// TwinCAT 3 PLC project PLC
// ProgramVersion: 3.1.4023.0
// libraries:
//   Tc2_Standard, * (Beckhoff Automation GmbH)
//   Tc2_System, * (Beckhoff Automation GmbH)
//   Tc3_Module, * (Beckhoff Automation GmbH)
// project tree:
//   DUTs/ ST_ControlBits.TcDUT, U_GatewayDataIn.TcDUT, ST_StatusBits.TcDUT, U_GatewayDataOut.TcDUT
//   / PlcTask.TcTTO
//   POUs/ MAIN.TcPOU
// real-time tasks:
//   TASK PlcTask: cycle T#2ms, priority 20, ADS port 350
// I/O:
//   DEVICE Device 1 (Profinet Device), AmsNetId 5.34.120.156.2.1
//     tcpniodevice [Beckhoff Automation TwinCAT PLC PROFINET I/O Device with I/Os, V2.32, 1 port diagnostic supported TwinCAT PN Device]
//       modules: Term 1 (DAP Module), Term 2 (32 Byte In- and Output)
//   DEVICE Device 2 (TC3 EIP Adapter), AmsNetId 5.34.120.156.3.1
//     Box 2 (TC EtherNet/IP Slave)
// variable links:
//   PLC Instance <-> Device 1 (Profinet Device)/tcpniodevice
//     PlcTask Inputs/MAIN.uPNIn.arBytes[{0..31}] <-> API/Term 2 (32 Byte In- and Output)/Subterm 4 (32 Byte In- and Output)/Inputs/1 Byte Output[{0..31}]  (32 links)
//     PlcTask Outputs/MAIN.uPNOut.arBytes[{0..31}] <-> API/Term 2 (32 Byte In- and Output)/Subterm 4 (32 Byte In- and Output)/Outputs/1 Byte Input[{0..31}]  (32 links)
//   PLC Instance <-> Device 2 (TC3 EIP Adapter)/Box 2 (TC EtherNet/IP Slave)
//     PlcTask Inputs/MAIN.uEIPIn.arBytes[{0..31}] <-> Assembly 1 (Input/Output)/Inputs/Var 139[{0..31}]  (32 links)
//     PlcTask Outputs/MAIN.uEIPOut.arBytes[{0..31}] <-> Assembly 1 (Input/Output)/Outputs/Var 172[{0..31}]  (32 links)

CONFIGURATION PLC
    RESOURCE PLC ON TwinCAT3
        TASK PlcTask(INTERVAL := T#2ms, PRIORITY := 20);
        PROGRAM MAIN WITH PlcTask : MAIN;
    END_RESOURCE
END_CONFIGURATION

// ---- DUTs/ST_ControlBits.TcDUT
TYPE ST_ControlBits :
STRUCT
	Start		:BIT;
	Stop		:BIT;
	Reset 		:BIT;
	bit4		:BIT;
	bit5		:BIT;
	bit6		:BIT;
	bit7		:BIT;
	bit8		:BIT;	
END_STRUCT
END_TYPE

// ---- DUTs/U_GatewayDataIn.TcDUT
TYPE U_GatewayDataIn :
UNION
	Status				:ST_StatusBits;
	arBytes 	AT%I*	:ARRAY[0..31] OF BYTE;
END_UNION
END_TYPE

// ---- DUTs/ST_StatusBits.TcDUT
TYPE ST_StatusBits :
STRUCT
	Starting	:BIT;
	Stopping	:BIT;
	Resting 	:BIT;
	Running		:BIT;
	bit5		:BIT;
	bit6		:BIT;
	bit7		:BIT;
	bit8		:BIT;	
END_STRUCT
END_TYPE

// ---- DUTs/U_GatewayDataOut.TcDUT
TYPE U_GatewayDataOut :
UNION
	Control				:ST_ControlBits;
	arBytes 	AT%Q*	:ARRAY[0..31] OF BYTE;	
END_UNION
END_TYPE

// ---- POUs/MAIN.TcPOU
PROGRAM MAIN
VAR
	GatewayIn						:ST_StatusBits;
	GatewayOut						:ST_ControlBits;

	uPNIn							:U_GatewayDataIn;
	uPNOut							:U_GatewayDataOut;	
	                            	
	uEIPIn							:U_GatewayDataIn;
	uEIPOut							:U_GatewayDataOut;	
		
    {IF defined (PN)}
        sVariantUsed                :STRING := 'PN';	
    {ELSIF defined (EIP)}
        sVariantUsed                :STRING := 'EIP';	
	{ELSIF defined (NoGateway)}	
		 sVariantUsed               :STRING := 'NoGateway';	
    {END_IF}

	Step							:INT;
	stepTimer						: TON := (PT := TIME#2S0MS);		
END_VAR

//Example of using the stucture of bits within the union
CASE Step OF
	0:
		GatewayOut.Start:=TRUE;
		stepTimer(IN:=TRUE);
		IF stepTimer.Q THEN
			GatewayOut.Start:=FALSE;
			stepTimer(IN:=FALSE);
	 		Step:=1;
		END_IF
	1:
		GatewayOut.Stop:=TRUE;
		stepTimer(IN:=TRUE);
		IF stepTimer.Q THEN
			GatewayOut.stop:=FALSE;
			stepTimer(IN:=FALSE);
	 		Step:=2;
		END_IF	
	2:
		GatewayOut.Reset:=TRUE;
		stepTimer(IN:=TRUE);
		IF stepTimer.Q THEN
			GatewayOut.Reset:=FALSE;
			stepTimer(IN:=FALSE);
	 		Step:=0;
		END_IF
	
END_CASE



//Map data based on current running varrient

{IF defined (PN)}
  	GatewayIn 			:=uPNIn.Status;
	uPNOut.Control		:=GatewayOut;
{ELSIF defined (EIP)}
  	GatewayIn 			:=uEIPIn.Status;
	uEIPOut.Control		:=GatewayOut;
{END_IF}

END_PROGRAM
